{attribute 'qualified_only'}
{attribute 'strict'}
{attribute 'to_string'}
TYPE E_OperatingMode :
(
    eMode_Manual := 0,
    eMode_Auto   := 1,
    eMode_Error  := 2
);
END_TYPE

(* stored: Version 1.1.0.1
   DUT E_OperatingMode: Id {78709dce-6b9f-418f-a790-0755ba495eaf} *)
